(* IEC 61131-3 sources: TCT_Proyect/ST_Generated, 3 files *)

(* ---- Assembly_line.st ---- *)
FUNCTION_BLOCK random_number
	VAR_INPUT
		IN : BOOL;
	END_VAR
	VAR
		M : BOOL;
		INIT : BOOL;
	END_VAR
	VAR_OUTPUT
		OUT : DINT;
	END_VAR

	IF INIT = 0 THEN
		{#include <stdio.h>}
		{#include <stdlib.h>}
		IN := 1;
	END_IF;
	IF M = 0 and IN = 1 THEN
		{SetFbVar(OUT,rand())}
	END_IF;
END_FUNCTION_BLOCK
PROGRAM tesis0
	VAR
		random : random_number;
		random_num : DINT;
		state : ARRAY [0..5] OF DINT;
		slt1 : ARRAY [0..8] OF DINT;
		slt2 : ARRAY [0..15] OF DINT;
		GD_OUT_4_G : ARRAY [0..2] OF BOOL;
		GD_OUT_7_G : ARRAY [0..2] OF BOOL;
		GD_OUT_8_G : ARRAY [0..2] OF BOOL;
		GD_OUT_5_G : ARRAY [0..3] OF BOOL;
		FE_LaP : F_TRIG;
		FE_BaP : F_TRIG;
		FE_PaL : F_TRIG;
		FE_Zag : F_TRIG;
		FE_Xag : F_TRIG;
	END_VAR
	VAR
		GD_OUT_12 AT %QX101.2 : BOOL;
 		GD_OUT_13 AT %QX101.3 : BOOL;
 		GD_OUT_2 AT %QX100.2 : BOOL;
		GD_OUT_3 AT %QX100.3 : BOOL;
		GD_OUT_4 AT %QX100.4 : BOOL;
		GD_OUT_5 AT %QX100.5 : BOOL;
		GD_OUT_6 AT %QX100.6 : BOOL;
		GD_OUT_7 AT %QX100.7 : BOOL;
		GD_OUT_8 AT %QX101.0 : BOOL;
		GD_OUT_9 AT %QX101.1 : BOOL;
		GD_IN_15 AT %IX100.15 : BOOL;
		GD_IN_2 AT %IX100.2 : BOOL;
		GD_IN_4 AT %IX100.4 : BOOL;
		GD_IN_3 AT %IX100.3 : BOOL;
		GD_IN_9 AT %IX101.1 : BOOL;
		GD_IN_5 AT %IX100.5 : BOOL;
		GD_IN_6 AT %IX100.6 : BOOL;
		GD_IN_7 AT %IX100.7 : BOOL;
		GD_IN_8 AT %IX101.0 : BOOL;
		GD_IN_10 AT %IX102.5 : BOOL;
		GD_IN_11 AT %IX102.6 : BOOL;
	END_VAR
	FE_LaP(CLK:= GD_IN_2);
	FE_BaP(CLK:= GD_IN_3);
	FE_PaL(CLK:= GD_IN_9);
	FE_Zag(CLK:= GD_IN_6);
	FE_Xag(CLK:= GD_IN_7);
	random(
		IN := True,
		OUT => random_num);
	IF state[0] = 0 & GD_IN_15 THEN
  		state[0] := 1;
  	ELSIF state[0] = 2 & FE_LaP.Q THEN
  		state[0] := 3;
  	ELSIF state[0] = 5 & GD_IN_4 THEN
  		state[0] := 6;
  	END_IF;

	IF state[1] = 0 & GD_IN_4 THEN
  		state[1] := 1;
  	ELSIF state[1] = 2 & GD_IN_4 THEN
  		state[1] := 3;
  	ELSIF state[1] = 4 & FE_Zag.Q THEN
  		state[1] := 6;
  	ELSIF state[1] = 5 & FE_Zag.Q THEN
  		state[1] := 7;
  	ELSIF state[1] = 12 & FE_Zag.Q THEN
  		state[1] := 14;
  	ELSIF state[1] = 13 & FE_Zag.Q THEN
  		state[1] := 15;
  	ELSIF state[1] = 16 & FE_Xag.Q THEN
  		state[1] := 18;
  	ELSIF state[1] = 17 & FE_Xag.Q THEN
  		state[1] := 19;
  	ELSIF state[1] = 20 & FE_Zag.Q THEN
  		state[1] := 22;
  	ELSIF state[1] = 21 & FE_Zag.Q THEN
  		state[1] := 23;
  	ELSIF state[1] = 26 & FE_Zag.Q THEN
  		state[1] := 28;
  	ELSIF state[1] = 27 & FE_Zag.Q THEN
  		state[1] := 29;
  	ELSIF state[1] = 30 & FE_Xag.Q THEN
  		state[1] := 0;
  	ELSIF state[1] = 31 & FE_Xag.Q THEN
  		state[1] := 2;
  	END_IF;

	IF state[2] = 2 & GD_IN_5 THEN
  		state[2] := 4;
  	ELSIF state[2] = 3 & GD_IN_5 THEN
  		state[2] := 5;
  	ELSIF state[2] = 6 & FE_Xag.Q THEN
  		state[2] := 8;
  	ELSIF state[2] = 7 & FE_Xag.Q THEN
  		state[2] := 9;
  	ELSIF state[2] = 10 & FE_Xag.Q THEN
  		state[2] := 12;
  	ELSIF state[2] = 11 & FE_Xag.Q THEN
  		state[2] := 16;
  	ELSIF state[2] = 13 & FE_Xag.Q THEN
  		state[2] := 20;
  	ELSIF state[2] = 14 & FE_Xag.Q THEN
  		state[2] := 17;
  	ELSIF state[2] = 15 & FE_Xag.Q THEN
  		state[2] := 19;
  	ELSIF state[2] = 18 & FE_Xag.Q THEN
  		state[2] := 25;
  	ELSIF state[2] = 21 & FE_Xag.Q THEN
  		state[2] := 24;
  	ELSIF state[2] = 22 & FE_Xag.Q THEN
  		state[2] := 27;
  	ELSIF state[2] = 22 & GD_IN_5 THEN
  		state[2] := 29;
  	ELSIF state[2] = 23 & FE_Xag.Q THEN
  		state[2] := 30;
  	ELSIF state[2] = 26 & FE_Xag.Q THEN
  		state[2] := 0;
  	ELSIF state[2] = 27 & GD_IN_5 THEN
  		state[2] := 34;
  	ELSIF state[2] = 28 & FE_Xag.Q THEN
  		state[2] := 32;
  	ELSIF state[2] = 28 & GD_IN_5 THEN
  		state[2] := 35;
  	ELSIF state[2] = 29 & FE_Xag.Q THEN
  		state[2] := 34;
  	ELSIF state[2] = 31 & FE_Xag.Q THEN
  		state[2] := 1;
  	ELSIF state[2] = 32 & GD_IN_5 THEN
  		state[2] := 37;
  	ELSIF state[2] = 33 & FE_Xag.Q THEN
  		state[2] := 2;
  	ELSIF state[2] = 33 & GD_IN_5 THEN
  		state[2] := 38;
  	ELSIF state[2] = 35 & FE_Xag.Q THEN
  		state[2] := 37;
  	ELSIF state[2] = 36 & FE_Xag.Q THEN
  		state[2] := 3;
  	ELSIF state[2] = 36 & GD_IN_5 THEN
  		state[2] := 39;
  	ELSIF state[2] = 38 & FE_Xag.Q THEN
  		state[2] := 4;
  	ELSIF state[2] = 39 & FE_Xag.Q THEN
  		state[2] := 5;
  	END_IF;

	IF state[3] = 0 & GD_IN_15 THEN
  		state[3] := 1;
  	ELSIF state[3] = 2 & FE_BaP.Q THEN
  		state[3] := 3;
  	ELSIF state[3] = 5 & GD_IN_5 THEN
  		state[3] := 6;
  	END_IF;

	IF state[4] = 3 & GD_IN_8 THEN
  		state[4] := 4;
  	ELSIF state[4] = 4 & FE_PaL.Q THEN
  		state[4] := 5;
  	END_IF;

	CASE state[0] OF
  		1:
  			GD_OUT_2 := 1;
		3:
  			GD_OUT_2 := 0;
  		4:
  			GD_OUT_4_G[0] := 1;
		6:
  			GD_OUT_4_G[0] := 0;
  	END_CASE;

	CASE state[1] OF
  		0:
  			GD_OUT_4_G[1] := 1;
		1:
  			CASE slt1[0] OF
  				0:
  					GD_OUT_4_G[1] := 1;
  				1:
  					GD_OUT_6 := 1;
  			END_CASE;
  			slt1[0] := (random_num + slt1[0]) MOD 2;
  			random_num := random_num - slt1[0];
 		3:
  			GD_OUT_6 := 1;
		4:
  			GD_OUT_4_G[1] := 1;
		6:
  			CASE slt1[1] OF
  				0:
  					GD_OUT_4_G[1] := 1;
  				1:
  					GD_OUT_7_G[0] := 1;
  			END_CASE;
  			slt1[1] := (random_num + slt1[1]) MOD 2;
  			random_num := random_num - slt1[1];
 		7:
  			GD_OUT_7_G[0] := 1;
		8:
  			GD_OUT_4_G[1] := 1;
		9:
  			GD_OUT_4_G[1] := 0;
  		10:
  			CASE slt1[2] OF
  				0:
  					GD_OUT_4_G[1] := 1;
  				1:
  					GD_OUT_6 := 0;
  			END_CASE;
  			slt1[2] := (random_num + slt1[2]) MOD 2;
  			random_num := random_num - slt1[2];
 		11:
  			GD_OUT_6 := 0;
  		12:
  			GD_OUT_4_G[1] := 1;
		14:
  			CASE slt1[3] OF
  				0:
  					GD_OUT_4_G[1] := 1;
  				1:
  					GD_OUT_8_G[0] := 1;
  			END_CASE;
  			slt1[3] := (random_num + slt1[3]) MOD 2;
  			random_num := random_num - slt1[3];
 		15:
  			GD_OUT_8_G[0] := 1;
		16:
  			GD_OUT_4_G[1] := 1;
		18:
  			CASE slt1[4] OF
  				0:
  					GD_OUT_4_G[1] := 1;
  				1:
  					GD_OUT_6 := 1;
  			END_CASE;
  			slt1[4] := (random_num + slt1[4]) MOD 2;
  			random_num := random_num - slt1[4];
 		19:
  			GD_OUT_6 := 1;
		20:
  			GD_OUT_4_G[1] := 1;
		22:
  			CASE slt1[5] OF
  				0:
  					GD_OUT_4_G[1] := 1;
  				1:
  					GD_OUT_7_G[0] := 0;
  			END_CASE;
  			slt1[5] := (random_num + slt1[5]) MOD 2;
  			random_num := random_num - slt1[5];
 		23:
  			GD_OUT_7_G[0] := 0;
  		24:
  			CASE slt1[6] OF
  				0:
  					GD_OUT_4_G[1] := 1;
  				1:
  					GD_OUT_6 := 0;
  			END_CASE;
  			slt1[6] := (random_num + slt1[6]) MOD 2;
  			random_num := random_num - slt1[6];
 		25:
  			GD_OUT_6 := 0;
  		26:
  			GD_OUT_4_G[1] := 1;
		28:
  			CASE slt1[7] OF
  				0:
  					GD_OUT_4_G[1] := 1;
  				1:
  					GD_OUT_8_G[0] := 0;
  			END_CASE;
  			slt1[7] := (random_num + slt1[7]) MOD 2;
  			random_num := random_num - slt1[7];
 		29:
  			GD_OUT_8_G[0] := 0;
  		30:
  			GD_OUT_4_G[1] := 1;
	END_CASE;

	CASE state[2] OF
  		0:
  			CASE slt2[0] OF
  				0:
  					GD_OUT_7_G[1] := 1;
  				1:
  					GD_OUT_5_G[0] := 1;
  			END_CASE;
  			slt2[0] := (random_num + slt2[0]) MOD 2;
  			random_num := random_num - slt2[0];
 		1:
  			GD_OUT_5_G[0] := 1;
		2:
  			GD_OUT_7_G[1] := 1;
		4:
  			CASE slt2[1] OF
  				0:
  					GD_OUT_7_G[1] := 1;
  				1:
  					GD_OUT_8_G[1] := 1;
  			END_CASE;
  			slt2[1] := (random_num + slt2[1]) MOD 2;
  			random_num := random_num - slt2[1];
 		5:
  			GD_OUT_8_G[1] := 1;
		6:
  			GD_OUT_7_G[1] := 1;
		7:
  			GD_OUT_7_G[1] := 0;
  		8:
  			CASE slt2[2] OF
  				0:
  					GD_OUT_7_G[1] := 1;
  				1:
  					GD_OUT_8_G[1] := 0;
  			END_CASE;
  			slt2[2] := (random_num + slt2[2]) MOD 2;
  			random_num := random_num - slt2[2];
 		9:
  			CASE slt2[3] OF
  				0:
  					GD_OUT_7_G[1] := 0;
  				1:
  					GD_OUT_8_G[1] := 0;
  			END_CASE;
  			slt2[3] := (random_num + slt2[3]) MOD 2;
  			random_num := random_num - slt2[3];
 		10:
  			CASE slt2[4] OF
  				0:
  					GD_OUT_7_G[1] := 1;
  				1:
  					GD_OUT_5_G[0] := 0;
  			END_CASE;
  			slt2[4] := (random_num + slt2[4]) MOD 2;
  			random_num := random_num - slt2[4];
 		11:
  			GD_OUT_7_G[1] := 1;
		12:
  			CASE slt2[5] OF
  				0:
  					GD_OUT_7_G[1] := 1;
  				1:
  					GD_OUT_8_G[1] := 0;
  				2:
  					GD_OUT_5_G[0] := 0;
  			END_CASE;
  			slt2[5] := (random_num + slt2[5]) MOD 3;
  			random_num := random_num - slt2[5];
 		13:
  			GD_OUT_7_G[1] := 0;
  		14:
  			GD_OUT_5_G[0] := 0;
  		15:
  			CASE slt2[6] OF
  				0:
  					GD_OUT_7_G[1] := 1;
  				1:
  					GD_OUT_5_G[0] := 1;
  			END_CASE;
  			slt2[6] := (random_num + slt2[6]) MOD 2;
  			random_num := random_num - slt2[6];
 		16:
  			GD_OUT_7_G[1] := 1;
		17:
  			CASE slt2[7] OF
  				0:
  					GD_OUT_8_G[1] := 0;
  				1:
  					GD_OUT_5_G[0] := 0;
  			END_CASE;
  			slt2[7] := (random_num + slt2[7]) MOD 2;
  			random_num := random_num - slt2[7];
 		18:
  			CASE slt2[8] OF
  				0:
  					GD_OUT_7_G[1] := 1;
  				1:
  					GD_OUT_5_G[0] := 0;
  			END_CASE;
  			slt2[8] := (random_num + slt2[8]) MOD 2;
  			random_num := random_num - slt2[8];
 		19:
  			CASE slt2[9] OF
  				0:
  					GD_OUT_7_G[1] := 1;
  				1:
  					GD_OUT_8_G[1] := 0;
  				2:
  					GD_OUT_5_G[0] := 1;
  			END_CASE;
  			slt2[9] := (random_num + slt2[9]) MOD 3;
  			random_num := random_num - slt2[9];
 		20:
  			GD_OUT_7_G[1] := 0;
  		21:
  			GD_OUT_5_G[0] := 1;
		22:
  			GD_OUT_7_G[1] := 1;
		23:
  			GD_OUT_5_G[0] := 0;
  		24:
  			CASE slt2[10] OF
  				0:
  					GD_OUT_8_G[1] := 0;
  				1:
  					GD_OUT_5_G[0] := 1;
  			END_CASE;
  			slt2[10] := (random_num + slt2[10]) MOD 2;
  			random_num := random_num - slt2[10];
 		25:
  			CASE slt2[11] OF
  				0:
  					GD_OUT_7_G[1] := 1;
  				1:
  					GD_OUT_5_G[0] := 0;
  			END_CASE;
  			slt2[11] := (random_num + slt2[11]) MOD 2;
  			random_num := random_num - slt2[11];
 		26:
  			CASE slt2[12] OF
  				0:
  					GD_OUT_7_G[1] := 1;
  				1:
  					GD_OUT_5_G[0] := 1;
  			END_CASE;
  			slt2[12] := (random_num + slt2[12]) MOD 2;
  			random_num := random_num - slt2[12];
 		27:
  			CASE slt2[13] OF
  				0:
  					GD_OUT_7_G[1] := 1;
  				1:
  					GD_OUT_8_G[1] := 0;
  			END_CASE;
  			slt2[13] := (random_num + slt2[13]) MOD 2;
  			random_num := random_num - slt2[13];
 		29:
  			GD_OUT_7_G[1] := 1;
		30:
  			GD_OUT_5_G[0] := 0;
  		31:
  			GD_OUT_5_G[0] := 1;
		32:
  			GD_OUT_8_G[1] := 0;
  		33:
  			GD_OUT_7_G[1] := 1;
		34:
  			CASE slt2[14] OF
  				0:
  					GD_OUT_7_G[1] := 1;
  				1:
  					GD_OUT_8_G[1] := 0;
  			END_CASE;
  			slt2[14] := (random_num + slt2[14]) MOD 2;
  			random_num := random_num - slt2[14];
 		37:
  			GD_OUT_8_G[1] := 0;
  		38:
  			GD_OUT_7_G[1] := 1;
	END_CASE;

	CASE state[3] OF
  		1:
  			GD_OUT_3 := 1;
		3:
  			GD_OUT_3 := 0;
  		4:
  			GD_OUT_5_G[1] := 1;
		6:
  			GD_OUT_5_G[1] := 0;
  	END_CASE;

	CASE state[4] OF
  		0:
  			GD_OUT_5_G[2] := 1;
		1:
  			GD_OUT_5_G[2] := 0;
  		2:
  			GD_OUT_9 := 1;
		5:
  			GD_OUT_9 := 0;
  	END_CASE;
	IF GD_OUT_4_G[0] <> GD_OUT_4_G[1] THEN
		GD_OUT_4_G[0] := GD_OUT_4;
		GD_OUT_4_G[1] := GD_OUT_4;
	END_IF;
	GD_OUT_4 := GD_OUT_4_G[0];
	IF GD_OUT_7_G[0] <> GD_OUT_7_G[1] THEN
		GD_OUT_7_G[0] := GD_OUT_7;
		GD_OUT_7_G[1] := GD_OUT_7;
	END_IF;
	GD_OUT_7 := GD_OUT_7_G[0];
	IF GD_OUT_8_G[0] <> GD_OUT_8_G[1] THEN
		GD_OUT_8_G[0] := GD_OUT_8;
		GD_OUT_8_G[1] := GD_OUT_8;
	END_IF;
	GD_OUT_8 := GD_OUT_8_G[0];
	IF (GD_OUT_5_G[0] <> GD_OUT_5_G[1]) OR (GD_OUT_5_G[1] <> GD_OUT_5_G[2]) THEN
		GD_OUT_5_G[0] := GD_OUT_5;
		GD_OUT_5_G[1] := GD_OUT_5;
		GD_OUT_5_G[2] := GD_OUT_5;
	END_IF;
	GD_OUT_5 := GD_OUT_5_G[0];
	IF state[0] = 1 & GD_OUT_2 THEN
  		state[0] := 2;
  	ELSIF state[0] = 3 & NOT GD_OUT_2 THEN
  		state[0] := 4;
  	ELSIF state[0] = 4 & GD_OUT_4 THEN
  		state[0] := 5;
  	ELSIF state[0] = 6 & NOT GD_OUT_4 THEN
  		state[0] := 1;
  	END_IF;

	IF state[1] = 0 & GD_OUT_4 THEN
  		state[1] := 2;
  	ELSIF state[1] = 1 & GD_OUT_4 THEN
  		state[1] := 3;
  	ELSIF state[1] = 1 & GD_OUT_6 THEN
  		state[1] := 4;
  	ELSIF state[1] = 3 & GD_OUT_6 THEN
  		state[1] := 5;
  	ELSIF state[1] = 4 & GD_OUT_4 THEN
  		state[1] := 5;
  	ELSIF state[1] = 6 & GD_OUT_4 THEN
  		state[1] := 7;
  	ELSIF state[1] = 6 & GD_OUT_7 THEN
  		state[1] := 8;
  	ELSIF state[1] = 7 & GD_OUT_7 THEN
  		state[1] := 9;
  	ELSIF state[1] = 8 & GD_OUT_4 THEN
  		state[1] := 9;
  	ELSIF state[1] = 9 & NOT GD_OUT_4 THEN
  		state[1] := 10;
  	ELSIF state[1] = 10 & GD_OUT_4 THEN
  		state[1] := 11;
  	ELSIF state[1] = 10 & NOT GD_OUT_6 THEN
  		state[1] := 12;
  	ELSIF state[1] = 11 & NOT GD_OUT_6 THEN
  		state[1] := 13;
  	ELSIF state[1] = 12 & GD_OUT_4 THEN
  		state[1] := 13;
  	ELSIF state[1] = 14 & GD_OUT_4 THEN
  		state[1] := 15;
  	ELSIF state[1] = 14 & GD_OUT_8 THEN
  		state[1] := 16;
  	ELSIF state[1] = 15 & GD_OUT_8 THEN
  		state[1] := 17;
  	ELSIF state[1] = 16 & GD_OUT_4 THEN
  		state[1] := 17;
  	ELSIF state[1] = 18 & GD_OUT_4 THEN
  		state[1] := 19;
  	ELSIF state[1] = 18 & GD_OUT_6 THEN
  		state[1] := 20;
  	ELSIF state[1] = 19 & GD_OUT_6 THEN
  		state[1] := 21;
  	ELSIF state[1] = 20 & GD_OUT_4 THEN
  		state[1] := 21;
  	ELSIF state[1] = 22 & GD_OUT_4 THEN
  		state[1] := 23;
  	ELSIF state[1] = 22 & NOT GD_OUT_7 THEN
  		state[1] := 24;
  	ELSIF state[1] = 23 & NOT GD_OUT_7 THEN
  		state[1] := 25;
  	ELSIF state[1] = 24 & GD_OUT_4 THEN
  		state[1] := 25;
  	ELSIF state[1] = 24 & NOT GD_OUT_6 THEN
  		state[1] := 26;
  	ELSIF state[1] = 25 & NOT GD_OUT_6 THEN
  		state[1] := 27;
  	ELSIF state[1] = 26 & GD_OUT_4 THEN
  		state[1] := 27;
  	ELSIF state[1] = 28 & GD_OUT_4 THEN
  		state[1] := 29;
  	ELSIF state[1] = 28 & NOT GD_OUT_8 THEN
  		state[1] := 30;
  	ELSIF state[1] = 29 & NOT GD_OUT_8 THEN
  		state[1] := 31;
  	ELSIF state[1] = 30 & GD_OUT_4 THEN
  		state[1] := 31;
  	END_IF;

	IF state[2] = 0 & GD_OUT_7 THEN
  		state[2] := 1;
  	ELSIF state[2] = 0 & GD_OUT_5 THEN
  		state[2] := 2;
  	ELSIF state[2] = 1 & GD_OUT_5 THEN
  		state[2] := 3;
  	ELSIF state[2] = 2 & GD_OUT_7 THEN
  		state[2] := 3;
  	ELSIF state[2] = 4 & GD_OUT_7 THEN
  		state[2] := 5;
  	ELSIF state[2] = 4 & GD_OUT_8 THEN
  		state[2] := 6;
  	ELSIF state[2] = 5 & GD_OUT_8 THEN
  		state[2] := 7;
  	ELSIF state[2] = 6 & GD_OUT_7 THEN
  		state[2] := 7;
  	ELSIF state[2] = 7 & NOT GD_OUT_7 THEN
  		state[2] := 10;
  	ELSIF state[2] = 8 & GD_OUT_7 THEN
  		state[2] := 9;
  	ELSIF state[2] = 8 & NOT GD_OUT_8 THEN
  		state[2] := 11;
  	ELSIF state[2] = 9 & NOT GD_OUT_7 THEN
  		state[2] := 12;
  	ELSIF state[2] = 9 & NOT GD_OUT_8 THEN
  		state[2] := 13;
  	ELSIF state[2] = 10 & GD_OUT_7 THEN
  		state[2] := 14;
  	ELSIF state[2] = 10 & NOT GD_OUT_5 THEN
  		state[2] := 15;
  	ELSIF state[2] = 11 & GD_OUT_7 THEN
  		state[2] := 13;
  	ELSIF state[2] = 12 & GD_OUT_7 THEN
  		state[2] := 17;
  	ELSIF state[2] = 12 & NOT GD_OUT_8 THEN
  		state[2] := 18;
  	ELSIF state[2] = 12 & NOT GD_OUT_5 THEN
  		state[2] := 19;
  	ELSIF state[2] = 13 & NOT GD_OUT_7 THEN
  		state[2] := 18;
  	ELSIF state[2] = 14 & NOT GD_OUT_5 THEN
  		state[2] := 21;
  	ELSIF state[2] = 15 & GD_OUT_7 THEN
  		state[2] := 21;
  	ELSIF state[2] = 15 & GD_OUT_5 THEN
  		state[2] := 22;
  	ELSIF state[2] = 16 & GD_OUT_7 THEN
  		state[2] := 20;
  	ELSIF state[2] = 17 & NOT GD_OUT_8 THEN
  		state[2] := 23;
  	ELSIF state[2] = 17 & NOT GD_OUT_5 THEN
  		state[2] := 24;
  	ELSIF state[2] = 18 & GD_OUT_7 THEN
  		state[2] := 23;
  	ELSIF state[2] = 18 & NOT GD_OUT_5 THEN
  		state[2] := 26;
  	ELSIF state[2] = 19 & GD_OUT_7 THEN
  		state[2] := 24;
  	ELSIF state[2] = 19 & NOT GD_OUT_8 THEN
  		state[2] := 26;
  	ELSIF state[2] = 19 & GD_OUT_5 THEN
  		state[2] := 27;
  	ELSIF state[2] = 20 & NOT GD_OUT_7 THEN
  		state[2] := 25;
  	ELSIF state[2] = 21 & GD_OUT_5 THEN
  		state[2] := 28;
  	ELSIF state[2] = 22 & GD_OUT_7 THEN
  		state[2] := 28;
  	ELSIF state[2] = 23 & NOT GD_OUT_5 THEN
  		state[2] := 31;
  	ELSIF state[2] = 24 & NOT GD_OUT_8 THEN
  		state[2] := 31;
  	ELSIF state[2] = 24 & GD_OUT_5 THEN
  		state[2] := 32;
  	ELSIF state[2] = 25 & GD_OUT_7 THEN
  		state[2] := 30;
  	ELSIF state[2] = 25 & NOT GD_OUT_5 THEN
  		state[2] := 0;
  	ELSIF state[2] = 26 & GD_OUT_7 THEN
  		state[2] := 31;
  	ELSIF state[2] = 26 & GD_OUT_5 THEN
  		state[2] := 33;
  	ELSIF state[2] = 27 & GD_OUT_7 THEN
  		state[2] := 32;
  	ELSIF state[2] = 27 & NOT GD_OUT_8 THEN
  		state[2] := 33;
  	ELSIF state[2] = 29 & GD_OUT_7 THEN
  		state[2] := 35;
  	ELSIF state[2] = 30 & NOT GD_OUT_5 THEN
  		state[2] := 1;
  	ELSIF state[2] = 31 & GD_OUT_5 THEN
  		state[2] := 36;
  	ELSIF state[2] = 32 & NOT GD_OUT_8 THEN
  		state[2] := 36;
  	ELSIF state[2] = 33 & GD_OUT_7 THEN
  		state[2] := 36;
  	ELSIF state[2] = 34 & GD_OUT_7 THEN
  		state[2] := 37;
  	ELSIF state[2] = 34 & NOT GD_OUT_8 THEN
  		state[2] := 38;
  	ELSIF state[2] = 37 & NOT GD_OUT_8 THEN
  		state[2] := 39;
  	ELSIF state[2] = 38 & GD_OUT_7 THEN
  		state[2] := 39;
  	END_IF;

	IF state[3] = 1 & GD_OUT_3 THEN
  		state[3] := 2;
  	ELSIF state[3] = 3 & NOT GD_OUT_3 THEN
  		state[3] := 4;
  	ELSIF state[3] = 4 & GD_OUT_5 THEN
  		state[3] := 5;
  	ELSIF state[3] = 6 & NOT GD_OUT_5 THEN
  		state[3] := 1;
  	END_IF;

	IF state[4] = 0 & GD_OUT_5 THEN
  		state[4] := 1;
  	ELSIF state[4] = 1 & NOT GD_OUT_5 THEN
  		state[4] := 2;
  	ELSIF state[4] = 2 & GD_OUT_9 THEN
  		state[4] := 3;
  	ELSIF state[4] = 5 & NOT GD_OUT_9 THEN
  		state[4] := 0;
  	END_IF;

	GD_OUT_12 := GD_IN_10;
 	GD_OUT_13 := GD_IN_11;

END_PROGRAM

CONFIGURATION Config0

	RESOURCE Res0 ON PLC
		TASK task0(INTERVAL := T#20ms,PRIORITY := 0);
		PROGRAM instance0 WITH task0 : tesis0;
	END_RESOURCE
END_CONFIGURATION

(* ---- Small_factory.st ---- *)
FUNCTION_BLOCK random_number
	VAR_INPUT
		IN : BOOL;
	END_VAR
	VAR
		M : BOOL;
		INIT : BOOL;
	END_VAR
	VAR_OUTPUT
		OUT : DINT;
	END_VAR

	IF INIT = 0 THEN
		{#include <stdio.h>}
		{#include <stdlib.h>}
		IN := 1;
	END_IF;
	IF M = 0 and IN = 1 THEN
		{SetFbVar(OUT,rand())}
	END_IF;
END_FUNCTION_BLOCK
PROGRAM tesis0
	VAR
		random : random_number;
		random_num : DINT;
		initial : BOOL;
		state : ARRAY [0..8] OF DINT;
		slt0 : ARRAY [0..2] OF DINT;
		FE_M1E : F_TRIG;
		FE_M2E : F_TRIG;
		FE_A : F_TRIG;
		FE_PL : F_TRIG;
		FE_PR : F_TRIG;
		INTERN_4 : BOOL;
		INTERN_5 : BOOL;
		INTERN_2 : BOOL;
		INTERN_3 : BOOL;
		INTERN_0 : BOOL;
		INTERN_1 : BOOL;
	END_VAR
	VAR
		GD_OUT_3 AT %QX100.3 : BOOL;
 		GD_OUT_8 AT %QX101.0 : BOOL;
 		GD_OUT_9 AT %QX101.1 : BOOL;
 		GD_OUT_0 AT %QX100.0 : BOOL;
		GD_OUT_1 AT %QX100.1 : BOOL;
		GD_IN_0 AT %IX100.0 : BOOL;
		GD_IN_1 AT %IX100.1 : BOOL;
		GD_IN_15 AT %IX100.5 : BOOL;
		GD_OUT_2 AT %QX100.2 : BOOL;
		GD_IN_2 AT %IX100.2 : BOOL;
		GD_OUT_4 AT %QX100.4 : BOOL;
		GD_IN_3 AT %IX100.3 : BOOL;
		GD_IN_4 AT %IX100.4 : BOOL;
		GD_OUT_5 AT %QX100.5 : BOOL;
		GD_OUT_6 AT %QX100.6 : BOOL;
		GD_IN_10 AT %IX101.0 : BOOL;
		GD_IN_11 AT %IX101.1 : BOOL;
		GD_IN_12 AT %IX101.2 : BOOL;
		GD_IN_13 AT %IX101.3 : BOOL;
		GD_OUT_10 AT %QX101.2 : BOOL;
		GD_OUT_11 AT %QX101.3 : BOOL;
	END_VAR
	FE_M1E(CLK:= GD_IN_0);
	FE_M2E(CLK:= GD_IN_1);
	FE_A(CLK:= GD_IN_2);
	FE_PL(CLK:= GD_IN_3);
	FE_PR(CLK:= GD_IN_4);
	random(
		IN := True,
		OUT => random_num);
	IF NOT initial THEN
		IF GD_IN_15 THEN
			initial := 1;
		END_IF;
	ELSIF initial THEN
		IF state[0] = 0 & GD_IN_15 THEN
	  		state[0] := 1;
	  	ELSIF state[0] = 2 & FE_PL.Q THEN
	  		state[0] := 3;
	  	ELSIF state[0] = 2 & NOT GD_IN_10 THEN
	  		state[0] := 4;
	  	ELSIF state[0] = 4 & NOT GD_IN_0 THEN
	  		state[0] := 1;
	  	ELSIF state[0] = 5 & FE_PL.Q THEN
	  		state[0] := 7;
	  	ELSIF state[0] = 5 & NOT GD_IN_10 THEN
	  		state[0] := 8;
	  	ELSIF state[0] = 6 & FE_M2E.Q THEN
	  		state[0] := 1;
	  	ELSIF state[0] = 6 & NOT GD_IN_11 THEN
	  		state[0] := 10;
	  	ELSIF state[0] = 8 & NOT GD_IN_0 THEN
	  		state[0] := 3;
	  	ELSIF state[0] = 9 & FE_M2E.Q THEN
	  		state[0] := 2;
	  	ELSIF state[0] = 9 & FE_PL.Q THEN
	  		state[0] := 11;
	  	ELSIF state[0] = 9 & NOT GD_IN_10 THEN
	  		state[0] := 12;
	  	ELSIF state[0] = 9 & NOT GD_IN_11 THEN
	  		state[0] := 13;
	  	ELSIF state[0] = 10 & FE_M2E.Q THEN
	  		state[0] := 14;
	  	ELSIF state[0] = 11 & FE_M2E.Q THEN
	  		state[0] := 3;
	  	ELSIF state[0] = 11 & NOT GD_IN_11 THEN
	  		state[0] := 16;
	  	ELSIF state[0] = 12 & FE_M2E.Q THEN
	  		state[0] := 4;
	  	ELSIF state[0] = 12 & NOT GD_IN_0 THEN
	  		state[0] := 6;
	  	ELSIF state[0] = 12 & NOT GD_IN_11 THEN
	  		state[0] := 17;
	  	ELSIF state[0] = 13 & FE_M2E.Q THEN
	  		state[0] := 18;
	  	ELSIF state[0] = 13 & FE_PL.Q THEN
	  		state[0] := 16;
	  	ELSIF state[0] = 13 & NOT GD_IN_10 THEN
	  		state[0] := 17;
	  	ELSIF state[0] = 15 & FE_M2E.Q THEN
	  		state[0] := 5;
	  	ELSIF state[0] = 15 & FE_PL.Q THEN
	  		state[0] := 20;
	  	ELSIF state[0] = 15 & NOT GD_IN_10 THEN
	  		state[0] := 19;
	  	ELSIF state[0] = 15 & NOT GD_IN_11 THEN
	  		state[0] := 21;
	  	ELSIF state[0] = 16 & FE_M2E.Q THEN
	  		state[0] := 22;
	  	ELSIF state[0] = 17 & FE_M2E.Q THEN
	  		state[0] := 23;
	  	ELSIF state[0] = 17 & NOT GD_IN_0 THEN
	  		state[0] := 10;
	  	ELSIF state[0] = 18 & FE_PL.Q THEN
	  		state[0] := 22;
	  	ELSIF state[0] = 18 & NOT GD_IN_10 THEN
	  		state[0] := 23;
	  	ELSIF state[0] = 19 & FE_M2E.Q THEN
	  		state[0] := 8;
	  	ELSIF state[0] = 19 & NOT GD_IN_0 THEN
	  		state[0] := 11;
	  	ELSIF state[0] = 19 & NOT GD_IN_11 THEN
	  		state[0] := 24;
	  	ELSIF state[0] = 20 & FE_M2E.Q THEN
	  		state[0] := 7;
	  	ELSIF state[0] = 20 & NOT GD_IN_11 THEN
	  		state[0] := 25;
	  	ELSIF state[0] = 21 & FE_M2E.Q THEN
	  		state[0] := 26;
	  	ELSIF state[0] = 21 & FE_PL.Q THEN
	  		state[0] := 25;
	  	ELSIF state[0] = 21 & NOT GD_IN_10 THEN
	  		state[0] := 24;
	  	ELSIF state[0] = 23 & NOT GD_IN_0 THEN
	  		state[0] := 14;
	  	ELSIF state[0] = 24 & FE_M2E.Q THEN
	  		state[0] := 28;
	  	ELSIF state[0] = 24 & NOT GD_IN_0 THEN
	  		state[0] := 16;
	  	ELSIF state[0] = 25 & FE_M2E.Q THEN
	  		state[0] := 29;
	  	ELSIF state[0] = 26 & FE_PL.Q THEN
	  		state[0] := 29;
	  	ELSIF state[0] = 26 & NOT GD_IN_10 THEN
	  		state[0] := 28;
	  	ELSIF state[0] = 27 & FE_M2E.Q THEN
	  		state[0] := 14;
	  	ELSIF state[0] = 27 & NOT GD_IN_11 THEN
	  		state[0] := 10;
	  	ELSIF state[0] = 28 & NOT GD_IN_0 THEN
	  		state[0] := 22;
	  	ELSIF state[0] = 30 & FE_M2E.Q THEN
	  		state[0] := 18;
	  	ELSIF state[0] = 30 & FE_PL.Q THEN
	  		state[0] := 32;
	  	ELSIF state[0] = 30 & NOT GD_IN_10 THEN
	  		state[0] := 31;
	  	ELSIF state[0] = 30 & NOT GD_IN_11 THEN
	  		state[0] := 13;
	  	ELSIF state[0] = 31 & FE_M2E.Q THEN
	  		state[0] := 23;
	  	ELSIF state[0] = 31 & NOT GD_IN_0 THEN
	  		state[0] := 27;
	  	ELSIF state[0] = 31 & NOT GD_IN_11 THEN
	  		state[0] := 17;
	  	ELSIF state[0] = 32 & FE_M2E.Q THEN
	  		state[0] := 22;
	  	ELSIF state[0] = 32 & NOT GD_IN_11 THEN
	  		state[0] := 16;
	  	ELSIF state[0] = 33 & FE_M2E.Q THEN
	  		state[0] := 26;
	  	ELSIF state[0] = 33 & FE_PL.Q THEN
	  		state[0] := 35;
	  	ELSIF state[0] = 33 & NOT GD_IN_10 THEN
	  		state[0] := 34;
	  	ELSIF state[0] = 33 & NOT GD_IN_11 THEN
	  		state[0] := 21;
	  	ELSIF state[0] = 34 & FE_M2E.Q THEN
	  		state[0] := 28;
	  	ELSIF state[0] = 34 & NOT GD_IN_0 THEN
	  		state[0] := 32;
	  	ELSIF state[0] = 34 & NOT GD_IN_11 THEN
	  		state[0] := 24;
	  	ELSIF state[0] = 35 & FE_M2E.Q THEN
	  		state[0] := 29;
	  	ELSIF state[0] = 35 & NOT GD_IN_11 THEN
	  		state[0] := 25;
	  	END_IF;

		IF state[1] = 0 & GD_OUT_0 THEN
	  		state[1] := 1;
	  	ELSIF state[1] = 1 & GD_IN_0 THEN
	  		state[1] := 2;
	  	ELSIF state[1] = 3 & FE_M1E.Q THEN
	  		state[1] := 0;
	  	END_IF;

		IF state[2] = 0 & GD_OUT_1 THEN
	  		state[2] := 1;
	  	ELSIF state[2] = 1 & GD_IN_1 THEN
	  		state[2] := 2;
	  	ELSIF state[2] = 3 & FE_M2E.Q THEN
	  		state[2] := 0;
	  	END_IF;

		IF state[3] = 0 & GD_IN_15 THEN
	  		state[3] := 1;
	  	ELSIF state[3] = 2 & FE_A.Q THEN
	  		state[3] := 3;
	  	ELSIF state[3] = 4 & FE_M1E.Q THEN
	  		state[3] := 1;
	  	END_IF;

		IF state[4] = 0 & GD_IN_0 THEN
	  		state[4] := 1;
	  	ELSIF state[4] = 1 & FE_M1E.Q THEN
	  		state[4] := 2;
	  	ELSIF state[4] = 3 & FE_PL.Q THEN
	  		state[4] := 4;
	  	ELSIF state[4] = 1 & NOT GD_IN_10 THEN
	  		state[4] := 5;
	  	ELSIF state[4] = 5 & FE_M1E.Q THEN
	  		state[4] := 0;
	  	END_IF;

		IF state[5] = 0 & GD_IN_15 THEN
	  		state[5] := 1;
	  	ELSIF state[5] = 1 & FE_M1E.Q THEN
	  		state[5] := 2;
	  	ELSIF state[5] = 3 & FE_PR.Q THEN
	  		state[5] := 4;
	  	ELSIF state[5] = 5 & FE_M2E.Q THEN
	  		state[5] := 2;
	  	ELSIF state[5] = 7 & FE_M2E.Q THEN
	  		state[5] := 2;
	  	ELSIF state[5] = 5 & FE_M1E.Q THEN
	  		state[5] := 6;
	  	ELSIF state[5] = 7 & FE_PL.Q THEN
	  		state[5] := 8;
	  	ELSIF state[5] = 1 & NOT GD_IN_10 THEN
	  		state[5] := 9;
	  	ELSIF state[5] = 9 & FE_M1E.Q THEN
	  		state[5] := 1;
	  	END_IF;

		IF state[6] = 0 & FE_M2E.Q THEN
	  		state[6] := 1;
	  	ELSIF state[6] = 2 & FE_PR.Q THEN
	  		state[6] := 3;
	  	END_IF;

		IF state[7] = 0 & NOT GD_IN_10 THEN
	  		state[7] := 1;
	  	ELSIF state[7] = 2 & GD_IN_12 THEN
	  		state[7] := 3;
	  	ELSIF state[7] = 5 & NOT GD_IN_0 THEN
	  		state[7] := 6;
	  	ELSIF state[7] = 0 & NOT GD_IN_11 THEN
	  		state[7] := 7;
	  	ELSIF state[7] = 8 & GD_IN_13 THEN
	  		state[7] := 9;
	  	ELSIF state[7] = 11 & FE_M2E.Q THEN
	  		state[7] := 12;
	  	ELSIF state[7] = 2 & NOT GD_IN_11 THEN
	  		state[7] := 13;
	  	ELSIF state[7] = 15 & GD_IN_13 THEN
	  		state[7] := 16;
	  	ELSIF state[7] = 18 & FE_M2E.Q THEN
	  		state[7] := 19;
	  	ELSIF state[7] = 8 & NOT GD_IN_10 THEN
	  		state[7] := 15;
	  	END_IF;

		CASE state[0] OF
	  		1:
	  			INTERN_0 := 1;
			3:
	  			CASE slt0[0] OF
	  				0:
	  					INTERN_0 := 1;
	  				1:
	  					INTERN_1 := 1;
	  			END_CASE;
	  			slt0[0] := (random_num + slt0[0]) MOD 2;
	  			random_num := random_num - slt0[0];
	 		5:
	  			INTERN_1 := 1;
			6:
	  			INTERN_0 := 1;
			7:
	  			INTERN_1 := 1;
			8:
	  			INTERN_1 := 1;
			10:
	  			INTERN_0 := 1;
			11:
	  			INTERN_0 := 1;
			14:
	  			INTERN_0 := 1;
			16:
	  			INTERN_0 := 1;
			22:
	  			CASE slt0[1] OF
	  				0:
	  					INTERN_0 := 1;
	  				1:
	  					INTERN_1 := 1;
	  			END_CASE;
	  			slt0[1] := (random_num + slt0[1]) MOD 2;
	  			random_num := random_num - slt0[1];
	 		26:
	  			INTERN_1 := 1;
			27:
	  			INTERN_0 := 1;
			28:
	  			INTERN_1 := 1;
			29:
	  			INTERN_1 := 1;
			32:
	  			INTERN_0 := 1;
		END_CASE;

		CASE state[1] OF
	  		2:
	  			GD_OUT_0 := 0;
	  	END_CASE;

		CASE state[2] OF
	  		2:
	  			GD_OUT_1 := 0;
	  	END_CASE;

		CASE state[3] OF
	  		1:
	  			GD_OUT_2 := 1;
			3:
	  			GD_OUT_2 := 0;
	  	END_CASE;

		CASE state[4] OF
	  		2:
	  			GD_OUT_5 := 1;
			4:
	  			GD_OUT_5 := 0;
	  	END_CASE;

		CASE state[5] OF
	  		2:
	  			GD_OUT_4 := 1;
			4:
	  			GD_OUT_4 := 0;
	  		6:
	  			GD_OUT_4 := 1;
			8:
	  			GD_OUT_4 := 0;
	  	END_CASE;

		CASE state[6] OF
	  		1:
	  			GD_OUT_6 := 0;
	  		3:
	  			GD_OUT_6 := 1;
		END_CASE;

		CASE state[7] OF
	  		1:
	  			INTERN_2 := 1;
			3:
	  			GD_OUT_10 := 1;
			4:
	  			INTERN_2 := 0;
	  		6:
	  			GD_OUT_10 := 0;
	  		7:
	  			INTERN_3 := 1;
			9:
	  			GD_OUT_11 := 1;
			10:
	  			INTERN_3 := 0;
	  		12:
	  			GD_OUT_11 := 0;
	  		13:
	  			INTERN_2 := 0;
	  		14:
	  			INTERN_3 := 1;
			16:
	  			GD_OUT_11 := 1;
			17:
	  			INTERN_3 := 0;
	  		19:
	  			GD_OUT_11 := 0;
	  	END_CASE;
		IF state[0] = 1 & INTERN_0 THEN
	  		state[0] := 2;
	  	ELSIF state[0] = 3 & INTERN_0 THEN
	  		state[0] := 5;
	  	ELSIF state[0] = 3 & INTERN_1 THEN
	  		state[0] := 6;
	  	ELSIF state[0] = 5 & INTERN_1 THEN
	  		state[0] := 9;
	  	ELSIF state[0] = 6 & INTERN_0 THEN
	  		state[0] := 9;
	  	ELSIF state[0] = 7 & INTERN_1 THEN
	  		state[0] := 11;
	  	ELSIF state[0] = 8 & INTERN_1 THEN
	  		state[0] := 12;
	  	ELSIF state[0] = 10 & INTERN_0 THEN
	  		state[0] := 13;
	  	ELSIF state[0] = 11 & INTERN_0 THEN
	  		state[0] := 15;
	  	ELSIF state[0] = 14 & INTERN_0 THEN
	  		state[0] := 18;
	  	ELSIF state[0] = 16 & INTERN_0 THEN
	  		state[0] := 21;
	  	ELSIF state[0] = 22 & INTERN_0 THEN
	  		state[0] := 26;
	  	ELSIF state[0] = 22 & INTERN_1 THEN
	  		state[0] := 27;
	  	ELSIF state[0] = 26 & INTERN_1 THEN
	  		state[0] := 30;
	  	ELSIF state[0] = 27 & INTERN_0 THEN
	  		state[0] := 30;
	  	ELSIF state[0] = 28 & INTERN_1 THEN
	  		state[0] := 31;
	  	ELSIF state[0] = 29 & INTERN_1 THEN
	  		state[0] := 32;
	  	ELSIF state[0] = 32 & INTERN_0 THEN
	  		state[0] := 33;
	  	END_IF;

		IF state[1] = 2 & NOT GD_OUT_0 THEN
	  		state[1] := 3;
	  	END_IF;

		IF state[2] = 2 & NOT GD_OUT_1 THEN
	  		state[2] := 3;
	  	END_IF;

		IF state[3] = 1 & GD_OUT_2 THEN
	  		state[3] := 2;
	  	ELSIF state[3] = 3 & NOT GD_OUT_2 THEN
	  		state[3] := 4;
	  	END_IF;

		IF state[4] = 2 & GD_OUT_5 THEN
	  		state[4] := 3;
	  	ELSIF state[4] = 4 & NOT GD_OUT_5 THEN
	  		state[4] := 0;
	  	END_IF;

		IF state[5] = 2 & GD_OUT_4 THEN
	  		state[5] := 3;
	  	ELSIF state[5] = 4 & NOT GD_OUT_4 THEN
	  		state[5] := 5;
	  	ELSIF state[5] = 6 & GD_OUT_4 THEN
	  		state[5] := 7;
	  	ELSIF state[5] = 8 & NOT GD_OUT_4 THEN
	  		state[5] := 5;
	  	END_IF;

		IF state[6] = 1 & NOT GD_OUT_6 THEN
	  		state[6] := 2;
	  	ELSIF state[6] = 3 & GD_OUT_6 THEN
	  		state[6] := 0;
	  	END_IF;

		IF state[7] = 1 & INTERN_2 THEN
	  		state[7] := 2;
	  	ELSIF state[7] = 3 & GD_OUT_10 THEN
	  		state[7] := 4;
	  	ELSIF state[7] = 4 & NOT INTERN_2 THEN
	  		state[7] := 5;
	  	ELSIF state[7] = 6 & NOT GD_OUT_10 THEN
	  		state[7] := 0;
	  	ELSIF state[7] = 7 & INTERN_3 THEN
	  		state[7] := 8;
	  	ELSIF state[7] = 9 & GD_OUT_11 THEN
	  		state[7] := 10;
	  	ELSIF state[7] = 10 & NOT INTERN_3 THEN
	  		state[7] := 11;
	  	ELSIF state[7] = 12 & NOT GD_OUT_11 THEN
	  		state[7] := 0;
	  	ELSIF state[7] = 13 & NOT INTERN_2 THEN
	  		state[7] := 14;
	  	ELSIF state[7] = 14 & INTERN_3 THEN
	  		state[7] := 15;
	  	ELSIF state[7] = 16 & GD_OUT_11 THEN
	  		state[7] := 17;
	  	ELSIF state[7] = 17 & NOT INTERN_3 THEN
	  		state[7] := 18;
	  	ELSIF state[7] = 19 & NOT GD_OUT_11 THEN
	  		state[7] := 1;
	  	END_IF;

		IF NOT GD_OUT_1 & INTERN_1 THEN
			GD_OUT_1 := 1;
		ELSIF GD_OUT_1 & INTERN_1 THEN
			INTERN_1 := 0;
		END_IF;
		IF NOT GD_OUT_0 & INTERN_0 THEN
			GD_OUT_0 := 1;
		ELSIF GD_OUT_0 & INTERN_0 THEN
			INTERN_0 := 0;
		END_IF;
		GD_OUT_3 := GD_OUT_2;
	 	GD_OUT_8 := NOT GD_IN_10;
	 	GD_OUT_9 := NOT GD_IN_11;

	END_IF;
END_PROGRAM

CONFIGURATION Config0

	RESOURCE Res0 ON PLC
		TASK task0(INTERVAL := T#20ms,PRIORITY := 0);
		PROGRAM instance0 WITH task0 : tesis0;
	END_RESOURCE
END_CONFIGURATION

(* ---- transfer_line.st ---- *)
FUNCTION_BLOCK random_number
	VAR_INPUT
		IN : BOOL;
	END_VAR
	VAR
		M : BOOL;
		INIT : BOOL;
	END_VAR
	VAR_OUTPUT
		OUT : DINT;
	END_VAR

	IF INIT = 0 THEN
		{#include <stdio.h>}
		{#include <stdlib.h>}
		IN := 1;
	END_IF;
	IF M = 0 and IN = 1 THEN
		{SetFbVar(OUT,rand())}
	END_IF;
END_FUNCTION_BLOCK
PROGRAM tesis0
	VAR
		random : random_number;
		random_num : DINT;
		initial : BOOL;
		state : ARRAY [0..9] OF DINT;
		aux : BOOL := 0;
		INTERN_1_C : ARRAY [0..1] OF BOOL;
		INTERN_3_C : ARRAY [0..1] OF BOOL;
		INTERN_5_C : ARRAY [0..1] OF BOOL;
		slt0 : ARRAY [0..2] OF DINT;
		INTERN_5_G : ARRAY [0..2] OF BOOL;
		INTERN_3_G : ARRAY [0..2] OF BOOL;
		INTERN_1_G : ARRAY [0..1] OF BOOL;
		RE_M1 : R_TRIG;
		FE_M2E : F_TRIG;
		FE_CP : F_TRIG;
		RE_CP : R_TRIG;
		FE_M1 : F_TRIG;
		FE_B1 : F_TRIG;
		FE_B1O : F_TRIG;
		FE_PO : F_TRIG;
		FE_PR : F_TRIG;
		FE_AT : F_TRIG;
		FE_MZ : F_TRIG;
		FE_RO : F_TRIG;
		INTERN_1 : BOOL;
		INTERN_3 : BOOL;
		INTERN_5 : BOOL;
	END_VAR
	VAR
		GD_OUT_1 AT %QX100.1 : BOOL;
 		GD_OUT_2 AT %QX100.2 : BOOL;
 		GD_OUT_3 AT %QX100.3 : BOOL;
 		GD_OUT_11 AT %QX101.3 : BOOL;
 		GD_OUT_12 AT %QX101.4 : BOOL;
 		GD_OUT_13 AT %QX101.5 : BOOL;
 		GD_OUT_14 AT %QX101.6 : BOOL;
 		GD_IN_0 AT %IX100.0 : BOOL;
		GD_IN_8 AT %IX101.0 : BOOL;
		GD_IN_1 AT %IX100.1 : BOOL;
		GD_IN_6 AT %IX100.6 : BOOL;
		GD_OUT_7 AT %QX100.7 : BOOL;
		GD_IN_7 AT %IX100.7 : BOOL;
		GD_OUT_4 AT %QX100.4 : BOOL;
		GD_IN_2 AT %IX100.2 : BOOL;
		GD_IN_3 AT %IX100.3 : BOOL;
		GD_OUT_5 AT %QX100.5 : BOOL;
		GD_OUT_6 AT %QX100.6 : BOOL;
		GD_IN_4 AT %IX100.4 : BOOL;
		GD_IN_5 AT %IX100.5 : BOOL;
		GD_OUT_8 AT %QX101.0 : BOOL;
		GD_OUT_9 AT %QX101.1 : BOOL;
		GD_OUT_10 AT %QX101.2 : BOOL;
		GD_IN_9 AT %IX101.1 : BOOL;
		GD_IN_11 AT %IX101.3 : BOOL;
		GD_IN_10 AT %IX101.2 : BOOL;
		GD_IN_12 AT %IX101.4 : BOOL;
		GD_IN_13 AT %IX101.5 : BOOL;
		GD_OUT_15 AT %QX101.7 : BOOL;
		GD_OUT_18 AT %QX102.2 : BOOL;
		GD_OUT_16 AT %QX102.0 : BOOL;
		GD_OUT_17 AT %QX102.1 : BOOL;
		GD_OUT_0 AT %QX100.0 : BOOL;
	END_VAR
	RE_M1(CLK:= GD_IN_1);
	FE_M2E(CLK:= GD_IN_6);
	FE_CP(CLK:= GD_IN_7);
	RE_CP(CLK:= GD_IN_7);
	FE_M1(CLK:= GD_IN_1);
	FE_B1(CLK:= GD_IN_3);
	FE_B1O(CLK:= GD_IN_5);
	FE_PO(CLK:= GD_IN_9);
	FE_PR(CLK:= GD_IN_11);
	FE_AT(CLK:= GD_IN_10);
	FE_MZ(CLK:= GD_IN_12);
	FE_RO(CLK:= GD_IN_13);
	random(
		IN := True,
		OUT => random_num);
	IF NOT initial THEN
		IF GD_IN_0 THEN
			initial := 1;
		END_IF;
	ELSIF initial THEN
		IF state[0] = 0 & GD_IN_0 THEN
	  		state[0] := 1;
	  	ELSIF state[0] = 2 & RE_M1.Q THEN
	  		state[0] := 4;
	  	ELSIF state[0] = 3 & FE_PR.Q THEN
	  		state[0] := 4;
	  	ELSIF state[0] = 3 & FE_PO.Q THEN
	  		state[0] := 1;
	  	ELSIF state[0] = 5 & RE_CP.Q THEN
	  		state[0] := 1;
	  	ELSIF state[0] = 6 & RE_M1.Q THEN
	  		state[0] := 8;
	  	ELSIF state[0] = 6 & RE_CP.Q THEN
	  		state[0] := 2;
	  	ELSIF state[0] = 7 & FE_PR.Q THEN
	  		state[0] := 8;
	  	ELSIF state[0] = 7 & RE_CP.Q THEN
	  		state[0] := 3;
	  	ELSIF state[0] = 7 & FE_PO.Q THEN
	  		state[0] := 5;
	  	ELSIF state[0] = 8 & RE_CP.Q THEN
	  		state[0] := 4;
	  	END_IF;

		IF state[1] = 1 & RE_CP.Q THEN
	  		state[1] := 2;
	  	ELSIF state[1] = 3 & FE_PR.Q THEN
	  		state[1] := 0;
	  	ELSIF state[1] = 3 & FE_PO.Q THEN
	  		state[1] := 0;
	  	ELSIF state[1] = 4 & FE_PR.Q THEN
	  		state[1] := 1;
	  	ELSIF state[1] = 4 & RE_CP.Q THEN
	  		state[1] := 5;
	  	ELSIF state[1] = 4 & FE_PO.Q THEN
	  		state[1] := 1;
	  	ELSIF state[1] = 5 & FE_PR.Q THEN
	  		state[1] := 2;
	  	ELSIF state[1] = 5 & FE_PO.Q THEN
	  		state[1] := 2;
	  	END_IF;

		IF state[2] = 0 & GD_OUT_0 THEN
	  		state[2] := 1;
	  	ELSIF state[2] = 0 & FE_M1.Q THEN
	  		state[2] := 2;
	  	ELSIF state[2] = 1 & FE_M1.Q THEN
	  		state[2] := 3;
	  	ELSIF state[2] = 2 & GD_OUT_0 THEN
	  		state[2] := 3;
	  	END_IF;

		IF state[3] = 0 & RE_M1.Q THEN
	  		state[3] := 1;
	  	ELSIF state[3] = 0 & FE_PR.Q THEN
	  		state[3] := 1;
	  	ELSIF state[3] = 2 & FE_B1.Q THEN
	  		state[3] := 3;
	  	ELSIF state[3] = 2 & FE_B1O.Q THEN
	  		state[3] := 4;
	  	ELSIF state[3] = 3 & FE_B1O.Q THEN
	  		state[3] := 5;
	  	ELSIF state[3] = 4 & FE_B1.Q THEN
	  		state[3] := 5;
	  	ELSIF state[3] = 4 & RE_M1.Q THEN
	  		state[3] := 7;
	  	ELSIF state[3] = 4 & FE_PR.Q THEN
	  		state[3] := 7;
	  	ELSIF state[3] = 5 & RE_M1.Q THEN
	  		state[3] := 8;
	  	ELSIF state[3] = 5 & FE_PR.Q THEN
	  		state[3] := 8;
	  	ELSIF state[3] = 6 & FE_B1O.Q THEN
	  		state[3] := 9;
	  	ELSIF state[3] = 7 & FE_B1.Q THEN
	  		state[3] := 8;
	  	ELSIF state[3] = 9 & RE_M1.Q THEN
	  		state[3] := 11;
	  	ELSIF state[3] = 9 & FE_PR.Q THEN
	  		state[3] := 11;
	  	ELSIF state[3] = 10 & GD_IN_2 THEN
	  		state[3] := 13;
	  	ELSIF state[3] = 10 & FE_B1O.Q THEN
	  		state[3] := 12;
	  	ELSIF state[3] = 12 & GD_IN_2 THEN
	  		state[3] := 15;
	  	ELSIF state[3] = 12 & RE_M1.Q THEN
	  		state[3] := 14;
	  	ELSIF state[3] = 12 & FE_PR.Q THEN
	  		state[3] := 14;
	  	ELSIF state[3] = 13 & FE_B1O.Q THEN
	  		state[3] := 15;
	  	ELSIF state[3] = 14 & GD_IN_2 THEN
	  		state[3] := 17;
	  	ELSIF state[3] = 15 & RE_M1.Q THEN
	  		state[3] := 17;
	  	ELSIF state[3] = 15 & FE_PR.Q THEN
	  		state[3] := 17;
	  	ELSIF state[3] = 16 & FE_B1O.Q THEN
	  		state[3] := 18;
	  	ELSIF state[3] = 18 & RE_M1.Q THEN
	  		state[3] := 20;
	  	ELSIF state[3] = 18 & FE_PR.Q THEN
	  		state[3] := 20;
	  	ELSIF state[3] = 19 & FE_B1O.Q THEN
	  		state[3] := 21;
	  	ELSIF state[3] = 21 & RE_M1.Q THEN
	  		state[3] := 23;
	  	ELSIF state[3] = 21 & FE_PR.Q THEN
	  		state[3] := 23;
	  	ELSIF state[3] = 22 & FE_B1O.Q THEN
	  		state[3] := 24;
	  	ELSIF state[3] = 24 & RE_M1.Q THEN
	  		state[3] := 26;
	  	ELSIF state[3] = 24 & FE_PR.Q THEN
	  		state[3] := 26;
	  	ELSIF state[3] = 25 & FE_B1O.Q THEN
	  		state[3] := 27;
	  	ELSIF state[3] = 27 & RE_M1.Q THEN
	  		state[3] := 28;
	  	ELSIF state[3] = 27 & FE_PR.Q THEN
	  		state[3] := 28;
	  	ELSIF state[3] = 29 & RE_M1.Q THEN
	  		state[3] := 30;
	  	ELSIF state[3] = 29 & FE_PR.Q THEN
	  		state[3] := 30;
	  	ELSIF state[3] = 31 & RE_M1.Q THEN
	  		state[3] := 32;
	  	ELSIF state[3] = 31 & FE_PR.Q THEN
	  		state[3] := 32;
	  	END_IF;

		IF state[4] = 0 & GD_OUT_7 THEN
	  		state[4] := 1;
	  	ELSIF state[4] = 1 & GD_IN_6 THEN
	  		state[4] := 2;
	  	ELSIF state[4] = 3 & FE_M2E.Q THEN
	  		state[4] := 0;
	  	END_IF;

		IF state[5] = 0 & GD_IN_6 THEN
	  		state[5] := 1;
	  	ELSIF state[5] = 1 & FE_M2E.Q THEN
	  		state[5] := 2;
	  	ELSIF state[5] = 3 & RE_CP.Q THEN
	  		state[5] := 4;
	  	END_IF;

		IF state[6] = 0 & GD_OUT_9 THEN
	  		state[6] := 1;
	  	ELSIF state[6] = 1 & FE_CP.Q THEN
	  		state[6] := 2;
	  	ELSIF state[6] = 2 & GD_IN_8 THEN
	  		state[6] := 3;
	  	ELSIF state[6] = 2 & NOT GD_IN_8 THEN
	  		state[6] := 4;
	  	ELSIF state[6] = 3 & FE_PO.Q THEN
	  		state[6] := 5;
	  	ELSIF state[6] = 6 & FE_AT.Q THEN
	  		state[6] := 7;
	  	END_IF;

		IF state[7] = 0 & FE_AT.Q THEN
	  		state[7] := 1;
	  	ELSIF state[7] = 2 & FE_MZ.Q THEN
	  		state[7] := 3;
	  	ELSIF state[7] = 5 & FE_MZ.Q THEN
	  		state[7] := 6;
	  	ELSIF state[7] = 7 & FE_RO.Q THEN
	  		state[7] := 8;
	  	ELSIF state[7] = 10 & FE_MZ.Q THEN
	  		state[7] := 11;
	  	ELSIF state[7] = 13 & FE_MZ.Q THEN
	  		state[7] := 14;
	  	ELSIF state[7] = 15 & FE_RO.Q THEN
	  		state[7] := 16;
	  	END_IF;

		CASE state[0] OF
	  		1:
	  			CASE slt0[0] OF
	  				0:
	  					INTERN_1_G[0] := 1;
	  				1:
	  					INTERN_5_G[0] := 1;
	  			END_CASE;
	  			slt0[0] := (random_num + slt0[0]) MOD 2;
	  			random_num := random_num - slt0[0];
	 		4:
	  			INTERN_3_G[0] := 1;
			5:
	  			CASE slt0[1] OF
	  				0:
	  					INTERN_1_G[0] := 1;
	  				1:
	  					INTERN_5_G[0] := 1;
	  			END_CASE;
	  			slt0[1] := (random_num + slt0[1]) MOD 2;
	  			random_num := random_num - slt0[1];
	 	END_CASE;

		CASE state[1] OF
	  		0:
	  			INTERN_3_G[1] := 1;
			2:
	  			INTERN_5_G[1] := 1;
			3:
	  			INTERN_3_G[1] := 1;
		END_CASE;

		CASE state[2] OF
	  		3:
	  			GD_OUT_0 := 0;
	  	END_CASE;

		CASE state[3] OF
	  		1:
	  			GD_OUT_5 := 1;
			3:
	  			GD_OUT_5 := 0;
	  		5:
	  			GD_OUT_5 := 0;
	  		6:
	  			GD_OUT_4 := 1;
			8:
	  			GD_OUT_5 := 0;
	  		9:
	  			GD_OUT_4 := 1;
			11:
	  			GD_OUT_4 := 1;
			13:
	  			GD_OUT_4 := 0;
	  		15:
	  			GD_OUT_4 := 0;
	  		16:
	  			GD_OUT_6 := 1;
			17:
	  			GD_OUT_4 := 0;
	  		18:
	  			GD_OUT_6 := 1;
			19:
	  			GD_IN_4 := 1;
			20:
	  			GD_OUT_6 := 1;
			21:
	  			GD_IN_4 := 1;
			22:
	  			GD_OUT_5 := 1;
			23:
	  			GD_IN_4 := 1;
			26:
	  			GD_OUT_5 := 1;
			27:
	  			GD_OUT_5 := 0;
	  		28:
	  			GD_OUT_5 := 0;
	  		29:
	  			GD_OUT_6 := 0;
	  		30:
	  			GD_OUT_6 := 0;
	  		31:
	  			GD_IN_4 := 1;
			32:
	  			GD_IN_4 := 1;
		END_CASE;

		CASE state[4] OF
	  		2:
	  			GD_OUT_7 := 0;
	  	END_CASE;

		CASE state[5] OF
	  		2:
	  			GD_OUT_8 := 1;
			4:
	  			GD_OUT_8 := 0;
	  	END_CASE;

		CASE state[6] OF
	  		4:
	  			GD_OUT_10 := 1;
			5:
	  			GD_OUT_9 := 0;
	  		7:
	  			GD_OUT_10 := 0;
	  		8:
	  			GD_OUT_9 := 0;
	  	END_CASE;

		CASE state[7] OF
	  		1:
	  			GD_OUT_15 := 1;
			3:
	  			GD_OUT_18 := 1;
			4:
	  			GD_OUT_15 := 0;
	  		6:
	  			GD_OUT_16 := 1;
			8:
	  			GD_OUT_16 := 0;
	  		9:
	  			GD_OUT_15 := 1;
			11:
	  			GD_OUT_18 := 0;
	  		12:
	  			GD_OUT_15 := 0;
	  		14:
	  			GD_OUT_17 := 1;
			16:
	  			GD_OUT_17 := 0;
	  	END_CASE;
		CASE state[8] OF
	  		0:
	  			INTERN_1_C[1] := 1;
				INTERN_3_C[1] := 1;
				INTERN_5_C[1] := 0;
			1:
	  			INTERN_1_C[1] := 0;
				INTERN_3_C[1] := 0;
				INTERN_5_C[1] := 1;
		END_CASE;
	  	IF INTERN_5_G[0] <> INTERN_5_G[1] THEN
			INTERN_5_G[0] := INTERN_5;
			INTERN_5_G[1] := INTERN_5;
		END_IF;
		aux := INTERN_5_G[0];
		IF aux XOR INTERN_5 THEN
			IF NOT aux & INTERN_5_C[0] THEN
				INTERN_5 := 0;
			ELSIF aux & INTERN_5_C[1] THEN
				INTERN_5 := 1;
			END_IF;
		END_IF;
		INTERN_5_G[0] := INTERN_5;
		IF INTERN_3_G[0] <> INTERN_3_G[1] THEN
			INTERN_3_G[0] := INTERN_3;
			INTERN_3_G[1] := INTERN_3;
		END_IF;
		aux := INTERN_3_G[0];
		IF aux XOR INTERN_3 THEN
			IF NOT aux & INTERN_3_C[0] THEN
				INTERN_3 := 0;
			ELSIF aux & INTERN_3_C[1] THEN
				INTERN_3 := 1;
			END_IF;
		END_IF;
		INTERN_3_G[0] := INTERN_3;

		aux := INTERN_1_G[0];
		IF aux XOR INTERN_1 THEN
			IF NOT aux & INTERN_1_C[0] THEN
				INTERN_1 := 0;
			ELSIF aux & INTERN_1_C[1] THEN
				INTERN_1 := 1;
			END_IF;
		END_IF;
		INTERN_1_G[0] := INTERN_1;
		IF state[8] = 0 & INTERN_3 THEN
	  		state[8] := 1;
	  	ELSIF state[8] = 1 & INTERN_5 THEN
	  		state[8] := 0;
	  	END_IF;
		IF state[0] = 1 & INTERN_1 THEN
	  		state[0] := 2;
	  	ELSIF state[0] = 1 & INTERN_5 THEN
	  		state[0] := 3;
	  	ELSIF state[0] = 4 & INTERN_3 THEN
	  		state[0] := 5;
	  	ELSIF state[0] = 5 & INTERN_1 THEN
	  		state[0] := 6;
	  	ELSIF state[0] = 5 & INTERN_5 THEN
	  		state[0] := 7;
	  	END_IF;

		IF state[1] = 0 & INTERN_3 THEN
	  		state[1] := 1;
	  	ELSIF state[1] = 2 & INTERN_5 THEN
	  		state[1] := 3;
	  	ELSIF state[1] = 3 & INTERN_3 THEN
	  		state[1] := 4;
	  	END_IF;

		IF state[2] = 3 & NOT GD_OUT_0 THEN
	  		state[2] := 0;
	  	END_IF;

		IF state[3] = 1 & GD_OUT_5 THEN
	  		state[3] := 2;
	  	ELSIF state[3] = 3 & NOT GD_OUT_5 THEN
	  		state[3] := 6;
	  	ELSIF state[3] = 5 & NOT GD_OUT_5 THEN
	  		state[3] := 9;
	  	ELSIF state[3] = 6 & GD_OUT_4 THEN
	  		state[3] := 10;
	  	ELSIF state[3] = 8 & NOT GD_OUT_5 THEN
	  		state[3] := 11;
	  	ELSIF state[3] = 9 & GD_OUT_4 THEN
	  		state[3] := 12;
	  	ELSIF state[3] = 11 & GD_OUT_4 THEN
	  		state[3] := 14;
	  	ELSIF state[3] = 13 & NOT GD_OUT_4 THEN
	  		state[3] := 16;
	  	ELSIF state[3] = 15 & NOT GD_OUT_4 THEN
	  		state[3] := 18;
	  	ELSIF state[3] = 16 & GD_OUT_6 THEN
	  		state[3] := 19;
	  	ELSIF state[3] = 17 & NOT GD_OUT_4 THEN
	  		state[3] := 20;
	  	ELSIF state[3] = 18 & GD_OUT_6 THEN
	  		state[3] := 21;
	  	ELSIF state[3] = 19 & GD_IN_4 THEN
	  		state[3] := 22;
	  	ELSIF state[3] = 20 & GD_OUT_6 THEN
	  		state[3] := 23;
	  	ELSIF state[3] = 21 & GD_IN_4 THEN
	  		state[3] := 24;
	  	ELSIF state[3] = 22 & GD_OUT_5 THEN
	  		state[3] := 25;
	  	ELSIF state[3] = 23 & GD_IN_4 THEN
	  		state[3] := 26;
	  	ELSIF state[3] = 26 & GD_OUT_5 THEN
	  		state[3] := 25;
	  	ELSIF state[3] = 27 & NOT GD_OUT_5 THEN
	  		state[3] := 29;
	  	ELSIF state[3] = 28 & NOT GD_OUT_5 THEN
	  		state[3] := 30;
	  	ELSIF state[3] = 29 & NOT GD_OUT_6 THEN
	  		state[3] := 31;
	  	ELSIF state[3] = 30 & NOT GD_OUT_6 THEN
	  		state[3] := 32;
	  	ELSIF state[3] = 31 & GD_IN_4 THEN
	  		state[3] := 0;
	  	ELSIF state[3] = 32 & GD_IN_4 THEN
	  		state[3] := 1;
	  	END_IF;

		IF state[4] = 2 & NOT GD_OUT_7 THEN
	  		state[4] := 3;
	  	END_IF;

		IF state[5] = 2 & GD_OUT_8 THEN
	  		state[5] := 3;
	  	ELSIF state[5] = 4 & NOT GD_OUT_8 THEN
	  		state[5] := 0;
	  	END_IF;

		IF state[6] = 4 & GD_OUT_10 THEN
	  		state[6] := 6;
	  	ELSIF state[6] = 5 & NOT GD_OUT_9 THEN
	  		state[6] := 0;
	  	ELSIF state[6] = 7 & NOT GD_OUT_10 THEN
	  		state[6] := 8;
	  	ELSIF state[6] = 8 & NOT GD_OUT_9 THEN
	  		state[6] := 0;
	  	END_IF;

		IF state[7] = 1 & GD_OUT_15 THEN
	  		state[7] := 2;
	  	ELSIF state[7] = 3 & GD_OUT_18 THEN
	  		state[7] := 4;
	  	ELSIF state[7] = 4 & NOT GD_OUT_15 THEN
	  		state[7] := 5;
	  	ELSIF state[7] = 6 & GD_OUT_16 THEN
	  		state[7] := 7;
	  	ELSIF state[7] = 8 & NOT GD_OUT_16 THEN
	  		state[7] := 9;
	  	ELSIF state[7] = 9 & GD_OUT_15 THEN
	  		state[7] := 10;
	  	ELSIF state[7] = 11 & NOT GD_OUT_18 THEN
	  		state[7] := 12;
	  	ELSIF state[7] = 12 & NOT GD_OUT_15 THEN
	  		state[7] := 13;
	  	ELSIF state[7] = 14 & GD_OUT_17 THEN
	  		state[7] := 15;
	  	ELSIF state[7] = 16 & NOT GD_OUT_17 THEN
	  		state[7] := 0;
	  	END_IF;

		IF NOT GD_OUT_0 & INTERN_1 THEN
			GD_OUT_0 := 1;
		ELSIF GD_OUT_0 & INTERN_1 THEN
			INTERN_1 := 0;
			INTERN_1_G[0] := 0;
	END_IF;
		IF NOT GD_OUT_7 & INTERN_3 THEN
			GD_OUT_7 := 1;
		ELSIF GD_OUT_7 & INTERN_3 THEN
			INTERN_3 := 0;
			INTERN_3_G[0] := 0;
	END_IF;
		IF NOT GD_OUT_9 & INTERN_5 THEN
			GD_OUT_9 := 1;
		ELSIF GD_OUT_9 & INTERN_5 THEN
			INTERN_5 := 0;
			INTERN_5_G[0] := 0;
	END_IF;
		GD_OUT_1 := GD_OUT_0;
	 	GD_OUT_2 := GD_OUT_0;
	 	GD_OUT_3 := GD_OUT_0;
	 	GD_OUT_11 := GD_OUT_10;
	 	GD_OUT_12 := GD_OUT_10;
	 	GD_OUT_13 := GD_OUT_10;
	 	GD_OUT_14 := GD_OUT_10;

	END_IF;
END_PROGRAM

CONFIGURATION Config0

	RESOURCE Res0 ON PLC
		TASK task0(INTERVAL := T#20ms,PRIORITY := 0);
		PROGRAM instance0 WITH task0 : tesis0;
	END_RESOURCE
END_CONFIGURATION
